{attribute 'strict'}
TYPE E_State :
(
	NotReady:=0,				//未准备好
	iRunning:=3,					//运行中
	Alarm:=2,					//报警中
	Ready:=1,					//准备好
	Done:=4          //工站完成
	
)UINT;
END_TYPE

(* stored: Version 1.1.0.1, ProductVersion 3.1.4024.9
   DUT E_State: Id {21135e33-2701-4434-aabd-cf22183955dd} *)
